// Mitsubishi GX Works2 project: auto forward-reverse control   PLC: FX1N/FX1NC

PROGRAM MAIN
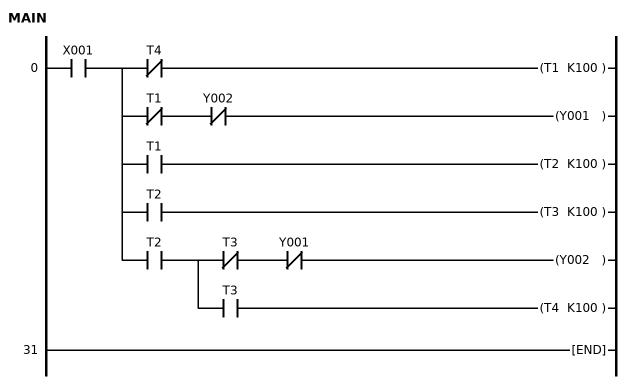
0     LD      X001
      MPS
      ANI     T4
      OUT     T1 K100
      MRD
      ANI     T1
      ANI     Y002
      OUT     Y001
      MRD
      AND     T1
      OUT     T2 K100
      MRD
      AND     T2
      OUT     T3 K100
      MPP
      AND     T2
      MPS
      ANI     T3
      ANI     Y001
      OUT     Y002
      MPP
      AND     T3
      OUT     T4 K100
31    END
END_PROGRAM
